# B&R Automation Studio project HealthCareDemo (part 2)

#### Router6D.fun - Exported functions and function blocks
```iecst
FUNCTION_BLOCK rl6dRouterMan (*Router manager*)
	VAR_INPUT
		Assembly : REFERENCE TO Mc6DAssemblyType; (*Assembly to manage shuttles on*)
		UserDataSize : UDINT; (*Size of the user data*)
		Enable : BOOL; (*Enable shuttle routing*)
	END_VAR
	VAR_OUTPUT
		Busy : BOOL; (*The function block is busy and must continue to be called*)
		Active : BOOL; (*The function block is active*)
		Error : BOOL; (*An error occurred*)
		ErrorID : DINT; (*Error that occurred*)
		Router : rl6dRouterType; (*Router handle*)
	END_VAR
	VAR
		Internal : rl6dRouterManInternalType; (*Internal data*)
	END_VAR
END_FUNCTION_BLOCK

FUNCTION_BLOCK rl6dRouterAddPathFromData (*Add a path from an array of positions*)
	VAR_INPUT
		Router : REFERENCE TO rl6dRouterType; (*Router to add path to*)
		DataAddress : UDINT; (*Pointer to array of rl6dPositionType*)
		DataSize : UDINT; (*Size of the array of positions in Bytes*)
		Name : STRING[255]; (*Name of the path*)
		Execute : BOOL; (*Add the path*)
	END_VAR
	VAR_OUTPUT
		Busy : BOOL; (*The function block is busy and must continue to be called*)
		Path : rl6dPathType; (*Path handle*)
		Done : BOOL; (*The path has been created*)
		Error : BOOL; (*An error occurred*)
		ErrorID : DINT; (*Error that occurred*)
	END_VAR
	VAR
		Internal : rl6dRouterAddPathInternalType; (*Internal data*)
	END_VAR
END_FUNCTION_BLOCK

FUNCTION_BLOCK rl6dPathGetData (*Get a path to an array of positions*)
	VAR_INPUT
		Path : REFERENCE TO rl6dPathType; (*Path handle*)
		DataAddress : UDINT; (*Pointer to array of rl6dPositionType*)
		DataSize : UDINT; (*Size of the array of positions in Bytes*)
		Execute : BOOL; (*Get the path*)
	END_VAR
	VAR_OUTPUT
		Busy : BOOL; (*The function block is busy and must continue to be called*)
		PathDataSize : UDINT; (*Actual size of path data*)
		Done : BOOL; (*The path has been created*)
		Error : BOOL; (*An error occurred*)
		ErrorID : DINT; (*Error that occurred*)
	END_VAR
	VAR
		Internal : rl6dGetPathInternalType; (*Internal data*)
	END_VAR
END_FUNCTION_BLOCK

FUNCTION_BLOCK rl6dRouterAddDestination (*Add a path from an array of positions*)
	VAR_INPUT
		Router : REFERENCE TO rl6dRouterType; (*Router to add destination to*)
		EntryPath : REFERENCE TO rl6dPathType; (*Optional reference to the destination entry path*)
		ExitPath : REFERENCE TO rl6dPathType; (*Optional reference to the destination exit path*)
		Position : rl6dPositionType; (*Position of the destination*)
		Name : STRING[255]; (*Name of the destination*)
		Execute : BOOL; (*Add the destination*)
	END_VAR
	VAR_OUTPUT
		Busy : BOOL; (*The function block is busy and must continue to be called*)
		Destination : rl6dDestinationType; (*Destination handle*)
		Done : BOOL; (*The destination has been created*)
		Error : BOOL; (*An error occurred*)
		ErrorID : DINT; (*Error that occurred*)
	END_VAR
	VAR
		Internal : rl6dRouterAddPathInternalType; (*Internal data*)
	END_VAR
END_FUNCTION_BLOCK

FUNCTION_BLOCK rl6dDestAddRecoveryPosFromData (*Add recovery positions from an array of positions*)
	VAR_INPUT
		Destination : REFERENCE TO rl6dDestinationType; (*Destination to add recovery points to*)
		DataAddress : UDINT; (*Pointer to array of rl6dPositionType*)
		DataSize : UDINT; (*Size of the array of positions in Bytes*)
		Execute : BOOL; (*Add the recovery points*)
	END_VAR
	VAR_OUTPUT
		Busy : BOOL; (*The function block is busy and must continue to be called*)
		Done : BOOL; (*The path has been created*)
		Error : BOOL; (*An error occurred*)
		ErrorID : DINT; (*Error that occurred*)
	END_VAR
	VAR
		Internal : rl6dDestAddRecPosInternalType; (*Internal data*)
	END_VAR
END_FUNCTION_BLOCK

FUNCTION_BLOCK rl6dDestinationSetWaypoint (*Set the waypoint of the destination*)
	VAR_INPUT
		Destination : REFERENCE TO rl6dDestinationType; (*Destination to set waypoint*)
		Waypoint : REFERENCE TO rl6dWaypointType; (*Waypoint to set*)
		Execute : BOOL; (*Set the next waypoint on a rising edge*)
	END_VAR
	VAR_OUTPUT
		Busy : BOOL; (*The function block is busy and must continue to be called*)
		Done : BOOL; (*The waypoint has been set*)
		Error : BOOL; (*An error occurred*)
		ErrorID : DINT; (*Error that occurred*)
	END_VAR
	VAR
		Internal : rl6dDestSetWaypntInternalType; (*Internal data*)
	END_VAR
END_FUNCTION_BLOCK

FUNCTION_BLOCK rl6dRouterAddWaypoint (*Add a waypoint from a position*)
	VAR_INPUT
		Router : REFERENCE TO rl6dRouterType; (*Router to add waypoint to*)
		Position : rl6dPositionType; (*Position of waypoint*)
		Name : STRING[255]; (*Name of waypoint*)
		Execute : BOOL; (*Add waypoint on rising edge*)
	END_VAR
	VAR_OUTPUT
		Busy : BOOL; (*The function block is busy and must continue to be called*)
		Waypoint : rl6dWaypointType; (*Waypoint handle*)
		Done : BOOL; (*The waypoint has been created*)
		Error : BOOL; (*An error occurred*)
		ErrorID : DINT; (*Error that occurred*)
	END_VAR
	VAR
		Internal : rl6dRouterAddWaypntInternalType; (*Internal data*)
	END_VAR
END_FUNCTION_BLOCK

FUNCTION_BLOCK rl6dWaypointAddDestination (*Add Destination to Waypoint*)
	VAR_INPUT
		Waypoint : REFERENCE TO rl6dWaypointType; (*Waypoint to add destination to*)
		Destination : REFERENCE TO rl6dDestinationType; (*Destination to add to waypoint*)
		DeparturePath : REFERENCE TO rl6dPathType; (*Optional departure path to follow when leaving waypoint for destination*)
		Execute : BOOL; (*Add the destination*)
	END_VAR
	VAR_OUTPUT
		Busy : BOOL; (*The function block is busy and must continue to be called*)
		Done : BOOL; (*The Destination has been added to the Waypoint*)
		Error : BOOL; (*An error occurred*)
		ErrorID : DINT; (*Error that occurred*)
	END_VAR
	VAR
		Internal : rl6dWaypointAddDestInternalType; (*Internal data*)
	END_VAR
END_FUNCTION_BLOCK

FUNCTION_BLOCK rl6dWaypointSetNextWaypoint (*Set the next waypoint of the target waypoint*)
	VAR_INPUT
		Waypoint : REFERENCE TO rl6dWaypointType; (*Waypoint to set next waypoint of*)
		NextWaypoint : REFERENCE TO rl6dWaypointType; (*Next waypoint*)
		Execute : BOOL; (*Set the next waypoint on a rising edge*)
	END_VAR
	VAR_OUTPUT
		Busy : BOOL; (*The function block is busy and must continue to be called*)
		Done : BOOL; (*The next waypoint has been set*)
		Error : BOOL; (*An error occurred*)
		ErrorID : DINT; (*Error that occurred*)
	END_VAR
	VAR
		Internal : rl6dWaypntSetWaypntInternalType; (*Internal data*)
	END_VAR
END_FUNCTION_BLOCK

FUNCTION_BLOCK rl6dRouterAddShFromAsm (*Add shuttles from the assembly*)
	VAR_INPUT
		Router : REFERENCE TO rl6dRouterType; (*Router to add shuttles from assembly to*)
		Execute : BOOL; (*Add shuttles*)
	END_VAR
	VAR_OUTPUT
		Busy : BOOL; (*The function block is busy and must continue to be called*)
		Done : BOOL; (*The shuttles have been added*)
		NumShuttles : UDINT; (*Number of shuttles found on the assembly*)
		Error : BOOL; (*An error occurred*)
		ErrorID : DINT; (*Error that occurred*)
	END_VAR
	VAR
		Internal : rl6dRtrAddShFromAsmInternalType; (*Internal data*)
	END_VAR
END_FUNCTION_BLOCK

FUNCTION_BLOCK rl6dRouterExecuteRecovery (*Execute recovery of shuttles*)
	VAR_INPUT
		Router : REFERENCE TO rl6dRouterType; (*Router to add shuttles from assembly to*)
		Velocity : REAL; (*Recovery Velocity*)
		Acceleration : REAL; (*Recovery Acceleration*)
		Mode : rl6dRecoverModeEnum; (*Mode to use when recovering*)
		Execute : BOOL; (*Add shuttles*)
	END_VAR
	VAR_OUTPUT
		Busy : BOOL; (*The function block is busy and must continue to be called*)
		Done : BOOL; (*The shuttles have been added*)
		Error : BOOL; (*An error occurred*)
		ErrorID : DINT; (*Error that occurred*)
	END_VAR
	VAR
		Internal : rl6dRtrAddShFromAsmInternalType; (*Internal data*)
	END_VAR
END_FUNCTION_BLOCK

FUNCTION_BLOCK rl6dDestinationMonitor (*Monitor destination for shuttles*)
	VAR_INPUT
		Destination : REFERENCE TO rl6dDestinationType; (*Destination to monitor*)
		Enable : BOOL; (*Enable monitoring*)
		AcknowledgeShuttle : BOOL; (*Acknowledge current shuttle*)
	END_VAR
	VAR_OUTPUT
		Busy : BOOL; (*The function block is busy and must continue to be called*)
		Valid : BOOL; (*Outputs are valid*)
		ShuttlePresent : BOOL; (*A shuttle is present at the destination*)
		ShuttleID : UINT; (*Shuttle ID*)
		RouterShuttle : rl6dShuttleType; (*Shuttle for use with router system*)
		Mc6DShuttle : Mc6DShuttleType; (*Shuttle for use with mapp 6D*)
		Error : BOOL; (*An error occurred*)
		ErrorID : DINT; (*Error that occurred*)
	END_VAR
	VAR
		Internal : rl6dDestinationMonInternalType; (*Internal data*)
	END_VAR
END_FUNCTION_BLOCK

FUNCTION_BLOCK rl6dShuttleMoveDestination (*Move shuttle to destination*)
	VAR_INPUT
		RouterShuttle : REFERENCE TO rl6dShuttleType; (*Shuttle to control*)
		Destination : REFERENCE TO rl6dDestinationType; (*Destination to move to*)
		Waypoint : REFERENCE TO rl6dWaypointType; (*Optional waypoint to override the waypoint specified by the previous destination*)
		Velocity : REAL; (*Velocity of shuttle movement*)
		Acceleration : REAL; (*Acceleration of shuttle movement*)
		Execute : BOOL; (*Start moving shuttle to destination*)
	END_VAR
	VAR_OUTPUT
		Busy : BOOL; (*The function block is busy and must continue to be called*)
		Active : BOOL; (*Move is active*)
		Aborted : BOOL; (*Move has been aborted*)
		Done : BOOL; (*Move has completed*)
		Error : BOOL; (*An error occurred*)
		ErrorID : DINT; (*Error that occurred*)
	END_VAR
	VAR
		Internal : rl6dShMoveDestInternalType; (*Internal data*)
	END_VAR
END_FUNCTION_BLOCK

FUNCTION_BLOCK rl6dShCopyUserData (*Copy shuttle user data asynchronously*)
	VAR_INPUT
		RouterShuttle : REFERENCE TO rl6dShuttleType; (*Shuttle to copy user data*)
		Mode : rl6dShCopyUserDataModeEnum; (*Mode of copy user data*)
		DataAddress : UDINT; (*Address of data to copy*)
		DataSize : UDINT; (*Start moving shuttle to destination*)
		Execute : BOOL; (*Copy user data*)
	END_VAR
	VAR_OUTPUT
		Busy : BOOL; (*The function block is busy and must continue to be called*)
		Done : BOOL; (*Move has completed*)
		SizeCopied : UDINT; (*Size of the data copied*)
		Error : BOOL; (*An error occurred*)
		ErrorID : DINT; (*Error that occurred*)
	END_VAR
	VAR
		Internal : rl6dShCopyUserDataInternalType; (*Internal Data*)
	END_VAR
END_FUNCTION_BLOCK

FUNCTION rl6dShCopyUserDataSync : DINT (*Copy shuttle user data synchronously*)
	VAR_INPUT
		RouterShuttle : rl6dShuttleType; (*Shuttle to copy user data*)
		Mode : rl6dShCopyUserDataModeEnum; (*Mode of copy*)
		DataAddress : UDINT; (*Data address*)
		DataSize : UDINT; (*Data size*)
	END_VAR
END_FUNCTION
```

#### CheckRef.hpp - Check Reference Headers
```cpp
#ifndef __RL6D_CHECK_REF_H__
#define __RL6D_CHECK_REF_H__

#include <Router.hpp>
#include <SemMan.hpp>
#include <Destination.hpp>
#include <DestinationIf.hpp>
#include <Path.hpp>
#include <Shuttle.hpp>
#include <ShuttleIf.hpp>

//Forward Declarations
class Router;
class SemMan;
class RouterSem;
class Destination;
class DestinationIf;
class Path;
class Shuttle;
class ShuttleIf;

DINT check_null_pointer(UDINT reference);

DINT check_router_reference(rl6dRouterType* reference);

DINT check_sem_man_reference(UDINT reference);

DINT check_router_sem_reference(UDINT reference);

DINT check_destination_reference(rl6dDestinationType* reference);

DINT check_destination_if_reference(UDINT reference);

DINT check_path_reference(rl6dPathType* reference);

DINT check_waypoint_reference(rl6dWaypointType* reference);

DINT check_shuttle_reference(rl6dShuttleType* reference);

DINT check_shuttle_if_reference(UDINT reference);

#endif
```

#### Logging.hpp - Logging Headers
```cpp
#ifndef __RL6D_LOGGING_H__
#define __RL6D_LOGGING_H__

#include <Router6D.h>
#include <string>
#include <cstring>

extern plcstring router_6d_log_name [];

bool log_routed_move_start(UINT shuttle, std::string destination);

bool log_direct_move_start(UINT shuttle, std::string destination);

bool log_destination_arrival(UINT shuttle, std::string destination);

bool log_destination_update(UINT shuttle, std::string destination);

bool log_path_start(UINT shuttle, std::string path);

bool log_waypoint_move(UINT shuttle, std::string waypoint);

bool log_routed_move_waypoint(UINT shuttle, std::string destination, std::string waypoint);

bool log_asm_get_sh_start(void);

bool log_asm_get_sh_done(UINT shuttles);

bool log_asm_recovery_start(rl6dRecoverModeEnum mode);

bool log_asm_recovery_done(void);

bool log_asm_sh_assignment(UINT shuttle, std::string destination);

bool log_sh_error(UINT shuttle, DINT error);

bool log_asm_get_sh_error(DINT error);

bool log_move_in_plane_error(DINT error);

#endif
```

#### Router.hpp - Router Headers
```cpp
#ifndef __RL6D_ROUTER_H__
#define __RL6D_ROUTER_H__

#include <memory>
#include <algorithm>
#include <cstring>

#include <CheckRef.hpp>
#include <Path.hpp>
#include <Waypoint.hpp>
#include <Shuttle.hpp>
#include <SemMan.hpp>
#include <Logging.hpp>

struct RouterCmd{
    bool add_sh_from_asm = 0;
    bool recover_shuttles = 0;
    rl6dRecoverModeEnum recover_shuttles_mode = rl6dRECOVER_MODE_BASIC;
    bool error_reset = 0;
};

struct RouterStatus{
    bool cmd_ready = 0;
    bool done = 0;
    bool error = 0;
    DINT error_id = 0;
};

struct ShDestAssignment{
    std::shared_ptr<Shuttle> shuttle;
    std::shared_ptr<Destination> destination;
};

/**
 \brief A Router manages shuttles to destinations
*/
class Router : public SemManBase{
    public:
    //! constructor for the Router
    Router(Mc6DAssemblyType* assembly, UDINT user_data_size);

    //! destructor for the Router
    ~Router(void);

    // members

    // methods
    //! Get the Router Type ID
    UDINT get_type_id(void);
    //! Create a new path
    std::shared_ptr<Path> create_path(std::string name, std::shared_ptr<RouterSem> router_sem);
    //! Delete a path
    void delete_path(std::shared_ptr<Path>);
    //! Get a path by name
    std::shared_ptr<Path> get_path_by_name(std::string name);
    //! Create a destination
    std::shared_ptr<Destination> create_destination(std::string name, std::shared_ptr<RouterSem> router_sem, rl6dPositionType position, std::shared_ptr<Path> path_in, std::shared_ptr<Path> path_out);
    //! Create a waypoint
    std::shared_ptr<Waypoint> create_waypoint(std::string name, std::shared_ptr<RouterSem> router_sem, rl6dPositionType position);
    //! Add a shuttle
    std::shared_ptr<Shuttle> add_shuttle(Mc6DShuttleType shuttle, std::shared_ptr<RouterSem> router_semaphore, UINT shuttle_id);
    //! Remove a shuttle
    void delete_shuttle(Mc6DShuttleType shuttle);
    //! Acquire path semaphore
    bool acquire_path_semaphore(void);
    //! Release path semaphore
    void release_path_semaphore(void);
    //! Acquire waypoint semaphore
    bool acquire_waypoint_semaphore(void);
    //! Release waypoint semaphore
    void release_waypoint_semaphore(void);
    //! Acquire shuttle semaphore
    bool acquire_shuttle_semaphore(void);
    //! Release shuttle semaphore
    void release_shuttle_semaphore(void);
    //! Acquire destination semaphore
    bool acquire_destination_semaphore(void);
    //! Release destination semaphore
    void release_destination_semaphore(void);
    //! Acquire command semaphore
    bool acquire_cmd_semaphore(void);
    //! Release command semaphore
    void release_cmd_semaphore(void);
    //! Set add shuttles from assembly
    void set_add_sh_from_asm();
    //! Reset add shuttles from assembly
    void reset_add_sh_from_asm(void);
    //! Set recover shuttles
    void set_recover_shuttles(rl6dRecoverModeEnum mode, REAL velocity, REAL acceleration);
    //! Reset recover shuttles
    void reset_recover_shuttles(void);
    //! Reset router errors
    void set_error_reset(void);
    //! get the number of shuttles found on the assembly
    UINT get_num_asm_sh(void);
    //! Get ready status
    bool get_cmd_ready(void);
    //! Get Done status
    bool get_done(void);
    //! Get error status
    bool get_error(void);
    //! Get error ID
    DINT get_error_id(void);
    //! Get initialized status
    bool get_initialized(void);
    //! Cyclic execution
    void cyclic(void);

    private:

    enum _state_enum
    {
        STATE_INIT,
        STATE_EVENT_LOG_CREATE,
        STATE_WAIT_SEM,
        STATE_CREATE_PATH_SEM,
        STATE_CREATE_WAYPOINT_SEM_READY,
        STATE_CREATE_WAYPOINT_SEM,
        STATE_CREATE_SHUTTLE_SEM_READY,
        STATE_CREATE_SHUTTLE_SEM,
        STATE_CREATE_DESTINATION_SEM_READY,
        STATE_CREATE_DESTINATION_SEM,
        STATE_CREATE_CMD_SEM_READY,
        STATE_CREATE_CMD_SEM,
        STATE_ACTIVE,
        STATE_ADD_SH_ASM,
        STATE_ADD_SH_ASM_SEM,
        STATE_ADD_SH_ASM_NEXT,
        STATE_ADD_SH_ASM_DONE,
        STATE_RECOVER_SHUTTLES_GET_DEST,
        STATE_RECOVER_SHUTTLES_GET_POS,
        STATE_RECOVER_SHUTTLES_ASSIGN,
        STATE_RECOVER_SHUTTLES,
        STATE_RECOVER_DESTINATION,
        STATE_RECOVER_DESTINATION_WAIT,
        STATE_RECOVER_SHUTTLES_DONE,
        STATE_ERROR
    };

    //! type identifier to ensure that pointer is valid
    UDINT _type_id = rl6dROUTER_TYPE_ID;
    //! state
    _state_enum _state = STATE_INIT;
    //! the list of paths that are part of the router
    std::vector<std::shared_ptr<Path>> _paths;
    //! the list of waypoints that are part of the router
    std::vector<std::shared_ptr<Waypoint>> _waypoints;
    //! the list of destinations that are part of the router
    std::vector<std::shared_ptr<Destination>> _destinations;
    //! the list of destinations to recover to
    std::vector<std::shared_ptr<Destination>> _recovery_destinations;
    //! current detination recovered shuttles are being assigned
    std::shared_ptr<Destination> _current_recovery_destination;
    //! current positions recovered shuttles are being assigned
    std::vector<rl6dPositionType> _current_recovery_positions;
    //! the list of shuttles that are part of the router
    std::vector<std::shared_ptr<Shuttle>> _shuttles;
    //! the list of shuttles to recover
    std::vector<std::shared_ptr<Shuttle>> _recovery_shuttles;
    //! current shuttle being recovered
    std::shared_ptr<Shuttle> _current_recovery_shuttle;
    //! current recovery index
    unsigned int _current_recovery_index = 0;
    //! current recovery position
    rl6dPositionType _current_recovery_position;
    //! the list of final recovery moves to make
    std::vector<ShDestAssignment> _shuttle_destination_assignment;
    //! current recovery shuttle interface
    std::shared_ptr<ShuttleIf> _current_recovery_shuttle_interface;
    //! the list of recovery shuttle interfaces
    std::vector<std::shared_ptr<ShuttleIf>> _shuttle_recovery_interfaces;
    //! Path semaphore
    std::shared_ptr<RouterSem> _path_semaphore;
    //! Waypoint semaphore
    std::shared_ptr<RouterSem> _waypoint_semaphore;
    //! Destination semaphore
    std::shared_ptr<RouterSem> _destination_semaphore;
    //! Shuttle semaphore
    std::shared_ptr<RouterSem> _shuttle_semaphore;
    //! Command semaphore
    std::shared_ptr<RouterSem> _command_semaphore;
    //! Router commands
    RouterCmd _cmd;
    //! Router status
    RouterStatus _status;
    //! Get shuttles from assembly
    struct MC_BR_AsmGetShuttle_Acp6D _asm_get_shuttle;
    //! Recover shuttles on assembly
    struct MC_BR_MoveInPlaneAsync_Acp6D _move_in_plane_async;
    //! Recorded number of shuttles remaining from assembly
    UDINT _old_remaining_count = 0;
    //! Recorded number of shuttles found on the assembly
    UDINT _asm_shuttles = 0;
    //! Newly created semaphore
    std::shared_ptr<RouterSem> _created_semaphore;
    //! Flag that initial semaphore creation is complete
    bool _router_sem_complete = 0;
    //! User data size for all shuttles
    UDINT _user_data_size;
    //! Initialization is complete
    bool _init_done = 0;
    //! Error
    bool _error = 0;
    //! Error ID
    DINT _error_id = ERR_OK;
    //EventLog Create
    struct ArEventLogCreate _ar_event_log_create;

};

#endif
```

#### SemMan.hpp - SemMan Headers
```cpp
#ifndef __RL6D_SEMMAN_H__
#define __RL6D_SEMMAN_H__

#include <memory>
#include <vector>
#include <algorithm>
#include <cstring>

#include <Router6D.h>

/**
 \brief A RouterSem contains a semaphore
*/
class RouterSem : public std::enable_shared_from_this<RouterSem>{
    public:
    //! constructor for the RouterSem
    RouterSem(UDINT semaphore);

    //! destructor for the RouterSem
    ~RouterSem(void);

    // members

    // methods
    //! Get the RouterSem Type ID
    UDINT get_type_id(void);
    //! Get the semaphore ident
    UDINT get_semaphore_ident(void);
    //! Delete this semaphore
    void set_delete(void);
    //! Check if this semaphore is to be deleted
    bool get_delete(void);
    //! Acquire the semaphore
    bool sem_acquire(void);
    //! Release the semaphore
    void sem_release(void);
    //! Get existing shared pointer
    std::shared_ptr<RouterSem> get_shared_ptr(void);

    private:

    //! type identifier to ensure that pointer is valid
    UDINT _type_id = rl6dROUTER_SEM_TYPE_ID;
    //! Semaphore to access
    UDINT _sem;
    //! Flag if this semaphore is to be deleted
    bool _delete = 0;

};

/**
 \brief A RouterSemBase gives a derived class the public methods and attributes to interface with the contained RouterSem
*/
class RouterSemBase{
    public:
    //! constructor for the RouterSem
    RouterSemBase(std::shared_ptr<RouterSem>);

    //! destructor for the RouterSem
    ~RouterSemBase(void);

    // members

    // methods
    //! Acquire the semaphore
    bool sem_acquire(void);
    //! Release the semaphore
    void sem_release(void);

    protected:

    //! Router semaphore
    std::shared_ptr<RouterSem> _router_semaphore;

};

struct SemManCmd{
    bool create_sem = 0;
    bool delete_all = 0;
};

struct SemManStatus{
    bool cmd_ready = 0;
    bool done = 0;
    bool error = 0;
    DINT error_id = 0;
};

/**
 \brief A SemMan mangages semaphores
*/
class SemMan{
    public:
    //! constructor for the SemMan
    SemMan(void);

    //! destructor for the SemMan
    ~SemMan(void);

    // members

    // methods
    //! Get the SemMan Type ID
    UDINT get_type_id(void);
    //! Create a new semaphore
    void set_create_sem(void);
    //! Reset creating a new semaphore
    void reset_create_sem(void);
    //! Return the newly created semaphore
    std::shared_ptr<RouterSem> get_created_sem(void);
    //! Get Done status
    bool get_done(void);
    //! Get Command Ready status
    bool get_cmd_ready(void);
    //! Get Error status
    bool get_error(void);
    //! Get Error ID
    DINT get_error_id(void);
    //! Delete a semaphore
    void delete_sem(UDINT);
    //! Acquire the semaphore to use other methods
    bool sem_acquire(void);
    //! Release the semaphore
    void sem_release(void);
    //! Get if the initialization is done
    bool get_initialized(void);
    //! Cyclic execution
    void cyclic(void);

    private:

    enum _state_enum
    {
        STATE_START,
        STATE_INIT,
        STATE_IDLE,
        STATE_CREATE_SEM,
        STATE_CREATE_SEM_DONE,
        STATE_DELETE_SEM,
        STATE_DELETE_ALL_SEM,
        STATE_DELETE_ALL_SEM_NEXT,
        STATE_DELETE_ALL_SEM_LAST,
        STATE_DELETE_ALL_SEM_DONE
    };

    //! type identifier to ensure that pointer is valid
    UDINT _type_id = rl6dSEM_MAN_TYPE_ID;
    //! state
    _state_enum _state = STATE_START;
    //! Semaphore to access manager
    UDINT _sem;
    //! Initialization is complete
    bool _init_done = 0;
    //! Commands
    SemManCmd _cmd;
    //! Status
    SemManStatus _status;
    //! Created semaphore
    std::shared_ptr<RouterSem> _created_semaphore;
    //! the list of semaphores being managed
    std::vector<std::shared_ptr<RouterSem>> _semaphores;
    //! Redo so that the iterator is not needed
    std::vector<std::shared_ptr<RouterSem>>::iterator _sem_iterator;
    //! semaphore generator
    struct SemCreate _create_semaphore;
    //! semaphore destructor
    struct SemDelete _delete_semaphore;

};

/**
 \brief A SemManBase gives a derived class the public methods and attributes to interface with the contained SemMan
*/
class SemManBase{
    public:
    //! constructor for the SemManBase
    SemManBase(void);

    //! destructor for the SemManBase
    ~SemManBase(void);

    // members

    // methods
    //! Create a new semaphore
    void set_create_sem(void);
    //! Reset creating a new semaphore
    void reset_create_sem(void);
    //! Return the newly created semaphore
    std::shared_ptr<RouterSem> get_created_sem(void);
    //! Get Done status
    bool get_sem_done(void);
    //! Get Command Ready status
    bool get_sem_cmd_ready(void);
    //! Get Error status
    bool get_sem_error(void);
    //! Get Error ID
    DINT get_sem_error_id(void);
    //! Acquire the semaphore to use other methods
    bool sem_acquire(void);
    //! Release the semaphore
    void sem_release(void);

    protected:

    //! SemMan
    SemMan _semaphore_manager;

};

#endif
```

#### Destination.hpp - Destination Headers
```cpp
#ifndef __RL6D_DESTINATION_H__
#define __RL6D_DESTINATION_H__

#include <memory>
#include <algorithm>
#include <string>
#include <vector>
#include <Router6D.h>

#include <Shuttle.hpp>
#include <Path.hpp>
#include <DestinationIf.hpp>
#include <Waypoint.hpp>

//Forward Declarations
class DestinationIf;
class Shuttle;
class Waypoint;

/**
 \brief A Destination is a position that a shuttle can travel to and can notify of its arrival
*/
class Destination: public RouterSemBase, public std::enable_shared_from_this<Destination>{
    public:
    //! constructor for the Destination
    Destination(std::string name, std::shared_ptr<RouterSem> router_sem);
    Destination(std::string name, std::shared_ptr<RouterSem> router_sem, rl6dPositionType position);
    Destination(std::string name, std::shared_ptr<RouterSem> router_sem, rl6dPositionType position, std::shared_ptr<Path> path_in, std::shared_ptr<Path> path_out);

    //! destructor for the Destination
    ~Destination(void);

    // members

    // methods
    //! Get the destination type ID
    UDINT get_type_id(void);
    //! Get the destination name
    std::string get_name(void);
    //! Get the destination position
    rl6dPositionType get_position(void);
    //! Get the recovery positions
    std::vector<rl6dPositionType> get_recovery_positions(void);
    //! Set the destination position
    void set_position(rl6dPositionType position);
    //! Get the destination path in
    std::shared_ptr<Path> get_path_in(void);
    //! Set the destination path in
    void set_path_in(std::shared_ptr<Path> path);
    //! Clear the destination path in
    void clear_path_in(void);
    //! Get the destination path out
    std::shared_ptr<Path> get_path_out(void);
    //! Set the destination path out
    void set_path_out(std::shared_ptr<Path> path);
    //! Clear the destination path out
    void clear_path_out(void);
    //! Add recovery position
    void add_recovery_position(rl6dPositionType position);
    //! Create interface
    std::shared_ptr<DestinationIf> create_interface(void);
    //! Set waypoint
    void set_waypoint(std::weak_ptr<Waypoint> waypoint);
    //! Get waypoint
    std::weak_ptr<Waypoint> get_waypoint(void);
    //! Reset waypoint
    void reset_waypoint(void);
    //! Set shuttle present
    void set_shuttle_present(std::weak_ptr<Shuttle> shuttle);
    //! Get existing shared pointer
    std::shared_ptr<Destination> get_shared_ptr(void);
    //! Cyclic runtime
    void cyclic(void);

    private:

    //! destination position
    rl6dPositionType _position;
    //! type identifier to ensure that pointer is valid
    UDINT _type_id = rl6dDESTINATION_TYPE_ID;
    //! name of the destination
    std::string _name;
    //! path in
    std::shared_ptr<Path> _path_in;
    //! path out
    std::shared_ptr<Path> _path_out;
    //! default waypoint
    std::weak_ptr<Waypoint> _waypoint;
    //! recovery points
    std::vector<rl6dPositionType> _recovery_positions;
    //! the list of destination interfaces that are part of the destination
    std::vector<std::shared_ptr<DestinationIf>> _interfaces;
    //! shuttle present at destination
    std::weak_ptr<Shuttle> _shuttle;
    //! shuttle present status
    bool _shuttle_present = 0;

};

#endif
```

#### DestinationIf.hpp - DestinationIf Headers
```cpp
#ifndef __RL6D_DESTINATION_IF_H__
#define __RL6D_DESTINATION_IF_H__

#include <memory>

#include <Router6D.h>
#include <Shuttle.hpp>

class Shuttle; //Forward Declaration

/**
 \brief A DestinationIf is an interface that can be monitored for shuttles
*/
class DestinationIf: public std::enable_shared_from_this<DestinationIf>{
    public:
    //! constructor for the DestinationIf
    DestinationIf(void);

    //! destructor for the DestinationIf
    ~DestinationIf(void);

    // members

    // methods
    //! Get the DestinationIf type ID
    UDINT get_type_id(void);
    //! Get existing shared pointer
    std::shared_ptr<DestinationIf> get_shared_ptr(void);
    //! Set shuttle status
    void set_shuttle_present(std::weak_ptr<Shuttle> shuttle);
    //! Get shuttle status
    bool shuttle_is_present(void);
    //! Get currently present shuttle
    std::weak_ptr<Shuttle> get_shuttle_present(void);
    //! Acknowledge shuttle present
    void acknowledge_shuttle(void);
    //! Set interface for deletion
    void set_delete(void);
    //! Check interface for deletion
    bool get_delete(void);

    private:

    //! type identifier to ensure that pointer is valid
    UDINT _type_id = rl6dDESTINATION_IF_TYPE_ID;
    //! Destination status of shuttle present
    bool _shuttle_present = 0;
    //! Shuttle present at Destination
    std::weak_ptr<Shuttle> _shuttle;
    //! Interface can be deleted
    bool _delete = 0;

};

#endif
```

#### Path.hpp - Path Headers
```cpp
#ifndef __RL6D_PATH_H__
#define __RL6D_PATH_H__

#include <string>
#include <vector>
#include <Router6D.h>
#include <SemMan.hpp>

/**
 \brief A Path is a vector of positions that the shuttle can travel along bust cannot leave
*/
class Path : public RouterSemBase, public std::enable_shared_from_this<Path>{
    public:
    //! constructor for the Path
    Path(std::string name, std::shared_ptr<RouterSem> router_sem);

    //! destructor for the Path
    ~Path(void);

    // members

    // methods
    //! Get the path type ID
    UDINT get_type_id(void);
    //! Get the path name
    std::string get_name(void);
    //! Add a position to the vector
    void add_position(rl6dPositionType position);
    //! Get position vector
    std::vector<rl6dPositionType> get_positions(void);
    //! Get existing shared pointer
    std::shared_ptr<Path> get_shared_ptr(void);

    private:

    //! the list of positions that are part of the path
    std::vector<rl6dPositionType> _positions;
    //! type identifier to ensure that pointer is valid
    UDINT _type_id = rl6dPATH_TYPE_ID;
    //! name of the path
    std::string _name;

};

#endif
```

#### Waypoint.hpp - Waypoint Headers
```cpp
#ifndef __RL6D_WAYPOINT_H__
#define __RL6D_WAYPOINT_H__

#include <Router6D.h>
#include <Path.hpp>
#include <Destination.hpp>

class Destination; //Forward declaration

struct WaypointDestination{
    std::shared_ptr<Destination> destination;
    std::shared_ptr<Path> departure_path;
};

/**
 \brief A Waypoint is a position that the shuttle will go through on its way to a destination, if defined
*/
class Waypoint : public RouterSemBase, public std::enable_shared_from_this<Waypoint>{
    public:
    //! constructor for the Waypoint
    Waypoint(std::string name, std::shared_ptr<RouterSem> router_sem);
    Waypoint(std::string name, std::shared_ptr<RouterSem> router_sem, rl6dPositionType position);

    //! destructor for the Waypoint
    ~Waypoint(void);

    // members

    // methods
    //! Get the waypoint type ID
    UDINT get_type_id(void);
    //! Get the waypoint name
    std::string get_name(void);

    //! Add an accessible destination to the waypoint
    void add_destination(std::shared_ptr<Destination> destination, std::shared_ptr<Path> departure_path);
    //! Check if a destination is accessible
    bool check_destination_accessible(std::shared_ptr<Destination> destination);
    //! Get destination departure path
    std::shared_ptr<Path> get_destination_departure_path(std::shared_ptr<Destination> destination);
    //! Get destination vector
    std::vector<WaypointDestination> get_destinations(void);
    //! Get position
    rl6dPositionType get_position(void);
    //! Get existing shared pointer
    std::shared_ptr<Waypoint> get_shared_ptr(void);
    //! Get next waypoint
    std::weak_ptr<Waypoint> get_next_waypoint(void);
    //! Set next waypoint
    void set_next_waypoint(std::weak_ptr<Waypoint> waypoint);
    //! Reset next waypoint
    void reset_next_waypoint(void);

    private:

    //! the next waypoint
    std::weak_ptr<Waypoint> _next_waypoint;
    //! the list of destinations accessible from the waypoint
    std::vector<WaypointDestination> _destinations;
    //! type identifier to ensure that pointer is valid
    UDINT _type_id = rl6dWAYPOINT_TYPE_ID;
    //! name of the waypoint
    std::string _name;
    //! position of the waypoint
    rl6dPositionType _position;

};

#endif
```

#### Shuttle.hpp - Shuttle Headers
```cpp
#ifndef __RL6D_SHUTTLE_H__
#define __RL6D_SHUTTLE_H__

#include <Router6D.h>
#include <McAcp6D.h>
#include <memory>
#include <vector>
#include <algorithm>
#include <cstring>

#include <Destination.hpp>
#include <Waypoint.hpp>
#include <Path.hpp>
#include <ShuttleIf.hpp>
#include <Logging.hpp>

class Destination; //Forward Declaration
class Waypoint; //Forward Declaration
class ShuttleIf; //Forward Declaration

struct ReadUserDataResult{
    char* value;
    UDINT size;
};

enum set_path_status_enum
{
    set_path_status_valid,
    set_path_status_invalid,
    set_path_status_wait_sem
};

enum routed_move_phase_enum
{
    ROUTED_MOVE_PHASE_EXIT_DEST_START,
    ROUTED_MOVE_PHASE_EXIT_DEST,
    ROUTED_MOVE_PHASE_WAYPOINT_START,
    ROUTED_MOVE_PHASE_WAYPOINT,
    ROUTED_MOVE_PHASE_DEPART_WAYPOINT_START,
    ROUTED_MOVE_PHASE_DEPART_WAYPOINT,
    ROUTED_MOVE_PHASE_ENTER_DEST_START,
    ROUTED_MOVE_PHASE_ENTER_DEST,
    ROUTED_MOVE_PHASE_DEST,
    ROUTED_MOVE_PHASE_ARRIVE
};

enum routed_move_event_enum
{
    ROUTED_MOVE_EVENT_NONE,
    ROUTED_MOVE_EVENT_PATH_START,
    ROUTED_MOVE_EVENT_WAYPOINT
};

struct RoutedMoveEvent{
    routed_move_event_enum event = ROUTED_MOVE_EVENT_NONE;
    std::shared_ptr<Path> path;
    std::weak_ptr<Waypoint> waypoint;
};

/**
 \brief A ShuttleRoutePositionGenerator outputs the positions on the shuttle route
*/
class ShuttleRoutePositionGenerator{
    public:
    //Constructor
    ShuttleRoutePositionGenerator(void);
    ShuttleRoutePositionGenerator(std::shared_ptr<Destination> previous_destination, std::shared_ptr<Destination> next_destination);
    ShuttleRoutePositionGenerator(std::shared_ptr<Destination> previous_destination, std::shared_ptr<Destination> next_destination, std::weak_ptr<Waypoint> route_waypoint);
    //Destructor
    ~ShuttleRoutePositionGenerator(void);

    //members

    //attributes
    rl6dPositionType position;
    RoutedMoveEvent event;

    //methods
    //! Increment the position along the route, return true if the route position has been incremented
    bool operator++(int);
    //! Update the destination
    void update_destination(std::shared_ptr<Destination> destination);
    void update_destination(std::shared_ptr<Destination> destination, std::weak_ptr<Waypoint> waypoint);
    //! Reset the position generator
    void reset(void);
    //! Get the current phase of the routed move
    routed_move_phase_enum get_phase(void);
    //! Get if the routed move is done
    bool get_done(void);

    private:

    //! Routing complete
    bool _done = 0;
    //! Set path, return set path status
    set_path_status_enum _set_path(std::shared_ptr<Path> path);
    //! Status of the exit path
    set_path_status_enum _exit_path_status = set_path_status_invalid;
    //! Status of the departure path
    set_path_status_enum _departure_path_status = set_path_status_invalid;
    //! Status of the entry path
    set_path_status_enum _entry_path_status = set_path_status_invalid;
    //! current waypoint
    std::weak_ptr<Waypoint> _current_waypoint;
    //! The phase of the routed motion
    routed_move_phase_enum _phase = ROUTED_MOVE_PHASE_EXIT_DEST_START;
    //! The previous destination the shuttle is going from
    std::shared_ptr<Destination>  _previous_destination;
    //! The next destination the shuttle is going to
    std::shared_ptr<Destination> _next_destination;
    //! The updated destination the shuttle needs to move to
    std::shared_ptr<Destination> _updated_destination;
    //! Route waypoint to use
    std::weak_ptr<Waypoint> _route_waypoint;
    //! path
    std::shared_ptr<Path> _path;
    //! path positions
    std::vector<rl6dPositionType> _path_positions;
    //! path iterator
    std::vector<rl6dPositionType>::iterator _path_iterator;
    //! Departure path
    std::shared_ptr<Path> _departure_path;

};

/**
 \brief A Shuttle controls an ACOPOS 6D shuttle
*/
class Shuttle : public RouterSemBase, public std::enable_shared_from_this<Shuttle>{
    public:
    //! constructor for the Shuttle
    Shuttle(Mc6DShuttleType shuttle, std::shared_ptr<RouterSem> router_sem, UDINT user_data_size, UINT _shuttle_id);

    //! destructor for the Shuttle
    ~Shuttle(void);

    // members

    // methods
    //! Get the shuttle type ID
    UDINT get_type_id(void);
    //! Get the shuttle ID
    UINT get_shuttle_id(void);
    //! Get the shuttle reference
    Mc6DShuttleType* get_shuttle_reference(void);
    //! Get the current destination
    std::shared_ptr<Destination> get_current_destination(void);
    //! Get the previous destination
    std::shared_ptr<Destination> get_previous_destination(void);
    //! Clear previous destination
    void clear_previous_destination(void);
    //! Create interface
    std::shared_ptr<ShuttleIf> create_interface(void);
    //! Get existing shared pointer
    std::shared_ptr<Shuttle> get_shared_ptr(void);
    //! Read User Data
    ReadUserDataResult read_user_data(void);
    //! Write User Data
    UDINT write_user_data(char* value, UDINT size);
    //! Cyclic runtime
    void cyclic(void);

    private:

    enum _state_enum
    {
        STATE_IDLE,
        STATE_ROUTED_MOVE_START,
        STATE_ROUTED_MOVE,
        STATE_ROUTED_MOVE_NEXT,
        STATE_DIRECT_MOVE,
    };

    //! Update shuttle interfaces
    bool _update_interfaces(void);
    //! Log events generated by the position generator
    void _log_event(RoutedMoveEvent event);
    //! type identifier to ensure that pointer is valid
    UDINT _type_id = rl6dSHUTTLE_TYPE_ID;
    //! 6D Shuttle ID
    UINT _shuttle_id;
    //! current interface
    std::shared_ptr<ShuttleIf> _current_interface;
    //! the list of shuttle interfaces that are part of the shuttle
    std::vector<std::shared_ptr<ShuttleIf>> _interfaces;
    //! The previous destination the shuttle is going from
    std::shared_ptr<Destination>  _previous_destination;
    //! The next destination the shuttle is going to
    std::shared_ptr<Destination> _next_destination;
    //! current state of cyclic execution
    _state_enum _state = STATE_IDLE;
    //! shuttle being managed
    Mc6DShuttleType _shuttle;
    //! move shuttle in plane
    struct MC_BR_MoveInPlane_Acp6D _move_in_plane;
    //! User Data
    std::unique_ptr<char[]> _user_data;
    //! User Data Size
    UDINT _user_data_size;
    //! Route position generator
    ShuttleRoutePositionGenerator _route_position_generator;
    //! Optional route waypoint
    std::weak_ptr<Waypoint> _optional_waypoint;

};

#endif
```

#### ShuttleIf.hpp - ShuttleIf Headers
```cpp
#ifndef __RL6D_SHUTTLE_IF_H__
#define __RL6D_SHUTTLE_IF_H__

#include <Router6D.h>

#include <Destination.hpp>
#include <Waypoint.hpp>

class Destination; //Forward Declaration
class Waypoint; //Forward Declaration

/**
 \brief A ShuttleIf is an interface that can be used to command shuttles
*/
class ShuttleIf : public std::enable_shared_from_this<ShuttleIf>{
    public:
    //! constructor for the ShuttleIf
    ShuttleIf(void);

    //! destructor for the ShuttleIf
    ~ShuttleIf(void);

    // members

    // methods
    //! Get the ShuttleIf type ID
    UDINT get_type_id(void);
    //! Issue move destination command
    void set_destination(std::shared_ptr<Destination> destination, REAL velocity, REAL acceleration);
    //! Issue move destination via waypoint command
    void set_destination_waypoint(std::shared_ptr<Destination> destination, std::weak_ptr<Waypoint> waypoint, REAL velocity, REAL acceleration);
    //! Check for move destination command
    bool get_destination_command(void);
    //! Issue move destination direct command
    void set_destination_direct(std::shared_ptr<Destination> destination, REAL velocity, REAL acceleration);
    //! Check for move destination direct command
    bool get_destination_direct_command(void);
    //! Get the destination commanded
    std::shared_ptr<Destination> get_destination(void);
    //! Get the waypoint commanded
    std::weak_ptr<Waypoint> get_waypoint(void);
    //! Set aborted status
    void set_aborted(void);
    //! Get aborted status
    bool get_aborted(void);
    //! Set error
    void set_error(DINT error);
    //! Get error status
    bool get_error(void);
    //! Get error id
    DINT get_error_id(void);
    //! Set move complete
    void set_move_done(void);
    //! Get move complete
    bool get_move_done(void);
    //! Set move active
    void set_move_active(void);
    //! Reset move active
    void reset_move_active(void);
    //! Get move active
    bool get_move_active(void);
    //! Set delete
    void set_delete(void);
    //! Get delete
    bool get_delete(void);
    //! Get velocity
    REAL get_velocity(void);
    //! Get acceleration
    REAL get_acceleration(void);
    //! Get existing shared pointer
    std::shared_ptr<ShuttleIf> get_shared_ptr(void);

    private:

    //! type identifier to ensure that pointer is valid
    UDINT _type_id = rl6dSHUTTLE_IF_TYPE_ID;
    //! Command Aborted
    bool _aborted = 0;
    //! Error
    bool _error = 0;
    //! Error ID
    DINT _error_id = 0;
    //! Move Destination
    bool _move_destination = 0;
    //! Move Destination Direct
    bool _move_destination_direct = 0;
    //! Destination
    std::shared_ptr<Destination> _destination;
    //! Route Waypoint
    std::weak_ptr<Waypoint> _waypoint;
    //! Velocity
    REAL _velocity;
    //! Acceleration
    REAL _acceleration;
    //! Move Done
    bool _move_done = 0;
    //! Move active
    bool _move_active = 0;
    //! Delete interface
    bool _delete = 0;

};

#endif
```

#### CheckRef.cpp - Check Reference Implementation
```cpp
#include "CheckRef.hpp"

DINT check_null_reference(UDINT reference){
    if(reference == 0){
        return rl6dERR_NULL_POINTER;
    }
    else{
        return ERR_OK;
    }
}

DINT check_router_reference(rl6dRouterType* reference){
    if(reference == nullptr){
        return rl6dERR_NULL_POINTER;
    }
    if(check_null_reference(reference->Ident) == ERR_OK){
        Router* router = reinterpret_cast<Router*>(reference->Ident);
        if(router->get_type_id() == rl6dROUTER_TYPE_ID){
            return ERR_OK;
        }
        else{
            return rl6dERR_ROUTER_INVALID;
        }
    }
    else{
        return rl6dERR_ROUTER_INVALID;
    }
}

DINT check_sem_man_reference(UDINT reference){
    DINT error;
    SemMan* sem_man;
    error = check_null_reference(reference);
    if(error == ERR_OK){
        sem_man = reinterpret_cast<SemMan*>(reference);
        if(sem_man->get_type_id() != rl6dSEM_MAN_TYPE_ID){
            error = rl6dERR_SEM_MAN_INVALID;
        }
    }
    return error;
}

DINT check_router_sem_reference(UDINT reference){
    DINT error;
    RouterSem* router_sem;
    error = check_null_reference(reference);
    if(error == ERR_OK){
        router_sem = reinterpret_cast<RouterSem*>(reference);
        if(router_sem->get_type_id() != rl6dROUTER_SEM_TYPE_ID){
            error = rl6dERR_ROUTER_SEM_INVALID;
        }
    }
    return error;
}

DINT check_destination_reference(rl6dDestinationType* reference){
    if(reference == nullptr){
        return rl6dERR_NULL_POINTER;
    }
    if(check_null_reference(reference->Ident) == ERR_OK){
        Destination* destination = reinterpret_cast<Destination*>(reference->Ident);
        if(destination->get_type_id() == rl6dDESTINATION_TYPE_ID){
            return ERR_OK;
        }
        else{
            return rl6dERR_DESTINATION_INVALID;
        }
    }
    else{
        return rl6dERR_DESTINATION_INVALID;
    }
}

DINT check_destination_if_reference(UDINT reference){
    DINT error;
    DestinationIf* destination_if;
    error = check_null_reference(reference);
    if(error == ERR_OK){
        destination_if = reinterpret_cast<DestinationIf*>(reference);
        if(destination_if->get_type_id() != rl6dDESTINATION_IF_TYPE_ID){
            error = rl6dERR_DESTINATION_IF_INVALID;
        }
    }
    return error;
}

DINT check_path_reference(rl6dPathType* reference){
    if(reference == nullptr){
        return rl6dERR_NULL_POINTER;
    }
    if(check_null_reference(reference->Ident) == ERR_OK){
        Path* path = reinterpret_cast<Path*>(reference->Ident);
        if(path->get_type_id() == rl6dPATH_TYPE_ID){
            return ERR_OK;
        }
        else{
            return rl6dERR_PATH_INVALID;
        }
    }
    else{
        return rl6dERR_PATH_INVALID;
    }
}

DINT check_waypoint_reference(rl6dWaypointType* reference){
    if(reference == nullptr){
        return rl6dERR_NULL_POINTER;
    }
    if(check_null_reference(reference->Ident) == ERR_OK){
        Waypoint* waypoint = reinterpret_cast<Waypoint*>(reference->Ident);
        if(waypoint->get_type_id() == rl6dWAYPOINT_TYPE_ID){
            return ERR_OK;
        }
        else{
            return rl6dERR_WAYPOINT_INVALID;
        }
    }
    else{
        return rl6dERR_WAYPOINT_INVALID;
    }
}

DINT check_shuttle_reference(rl6dShuttleType* reference){
    if(reference == nullptr){
        return rl6dERR_NULL_POINTER;
    }
    if(check_null_reference(reference->Ident) == ERR_OK){
        Shuttle* shuttle = reinterpret_cast<Shuttle*>(reference->Ident);
        if(shuttle->get_type_id() == rl6dSHUTTLE_TYPE_ID){
            return ERR_OK;
        }
        else{
            return rl6dERR_SHUTTLE_INVALID;
        }
    }
    else{
        return rl6dERR_SHUTTLE_INVALID;
    }
}

DINT check_shuttle_if_reference(UDINT reference){
    DINT error;
    ShuttleIf* shuttle_if;
    error = check_null_reference(reference);
    if(error == ERR_OK){
        shuttle_if = reinterpret_cast<ShuttleIf*>(reference);
        if(shuttle_if->get_type_id() != rl6dSHUTTLE_IF_TYPE_ID){
            error = rl6dERR_SHUTTLE_IF_INVALID;
        }
    }
    return error;
}
```

#### Logging.cpp - Logging Implementation
```cpp
#include "logging.hpp"

plcstring router_6d_log_name [] = "rl6dLog";

UDINT rl6d_log_buffer_min_size = 40;
UDINT rl6d_log_buffer_size_udint = 5;

bool log_routed_move_start(UINT shuttle, std::string destination){

    struct ArEventLogGetIdent get_ident;
    struct ArEventLogWrite write;

    bool status;
    UDINT buffer_size = destination.length() + 1;
    buffer_size += rl6d_log_buffer_min_size + rl6d_log_buffer_size_udint;
    char buffer [buffer_size];
    status = ArEventLogAddDataInit(reinterpret_cast<UDINT>(buffer), buffer_size, arEVENTLOG_ADDFORMAT_CODED);
    if(status){
        status = ArEventLogAddDataUdint(reinterpret_cast<UDINT>(buffer), buffer_size, shuttle);
    }
    if(status){
        status = ArEventLogAddDataString(reinterpret_cast<UDINT>(buffer), buffer_size, reinterpret_cast<UDINT>(destination.c_str()));
    }

    std::memset(&get_ident, 0, sizeof(get_ident));

    std::strcpy(get_ident.Name, router_6d_log_name);
    get_ident.Execute = 0;

    if(status){
        ArEventLogGetIdent(&get_ident);
        get_ident.Execute = 1;
        ArEventLogGetIdent(&get_ident);
        status = get_ident.Done;
        if(!status){
            get_ident.Execute = 0;
            ArEventLogGetIdent(&get_ident);
        }
    }

    std::memset(&write, 0, sizeof(write));

    std::string object = "RouterShuttle";
    object.append(std::to_string(shuttle));

    write.Ident = get_ident.Ident;
    std::strcpy(reinterpret_cast<char*>(&write.ObjectID), object.c_str());
    write.EventID = rl6dINFO_ROUTED_MOVE_START;
    write.AddData = reinterpret_cast<UDINT>(buffer);
    write.AddDataFormat = arEVENTLOG_ADDFORMAT_CODED;
    write.Execute = 0;

    if(status){
        ArEventLogWrite(&write);
        write.Execute = 1;
        ArEventLogWrite(&write);
        status = write.Done;
        write.Execute = 0;
        ArEventLogWrite(&write);
        get_ident.Execute = 0;
        ArEventLogGetIdent(&get_ident);
    }

    return status;

}

bool log_direct_move_start(UINT shuttle, std::string destination){

    struct ArEventLogGetIdent get_ident;
    struct ArEventLogWrite write;

    bool status;
    UDINT buffer_size = destination.length() + 1;
    buffer_size += rl6d_log_buffer_min_size + rl6d_log_buffer_size_udint;
    char buffer [buffer_size];
    status = ArEventLogAddDataInit(reinterpret_cast<UDINT>(buffer), buffer_size, arEVENTLOG_ADDFORMAT_CODED);
    if(status){
        status = ArEventLogAddDataUdint(reinterpret_cast<UDINT>(buffer), buffer_size, shuttle);
    }
    if(status){
        status = ArEventLogAddDataString(reinterpret_cast<UDINT>(buffer), buffer_size, reinterpret_cast<UDINT>(destination.c_str()));
    }

    std::memset(&get_ident, 0, sizeof(get_ident));

    std::strcpy(get_ident.Name, router_6d_log_name);
    get_ident.Execute = 0;

    if(status){
        ArEventLogGetIdent(&get_ident);
        get_ident.Execute = 1;
        ArEventLogGetIdent(&get_ident);
        status = get_ident.Done;
        if(!status){
            get_ident.Execute = 0;
            ArEventLogGetIdent(&get_ident);
        }
    }

    std::memset(&write, 0, sizeof(write));

    std::string object = "RouterShuttle";
    object.append(std::to_string(shuttle));

    write.Ident = get_ident.Ident;
    std::strcpy(reinterpret_cast<char*>(&write.ObjectID), object.c_str());
    write.EventID = rl6dINFO_DIRECT_MOVE_START;
    write.AddData = reinterpret_cast<UDINT>(buffer);
    write.AddDataFormat = arEVENTLOG_ADDFORMAT_CODED;
    write.Execute = 0;

    if(status){
        ArEventLogWrite(&write);
        write.Execute = 1;
        ArEventLogWrite(&write);
        status = write.Done;
        write.Execute = 0;
        ArEventLogWrite(&write);
        get_ident.Execute = 0;
        ArEventLogGetIdent(&get_ident);
    }

    return status;

}

bool log_destination_arrival(UINT shuttle, std::string destination){

    struct ArEventLogGetIdent get_ident;
    struct ArEventLogWrite write;

    bool status;
    UDINT buffer_size = destination.length() + 1;
    buffer_size += rl6d_log_buffer_min_size + rl6d_log_buffer_size_udint;
    char buffer [buffer_size];
    status = ArEventLogAddDataInit(reinterpret_cast<UDINT>(buffer), buffer_size, arEVENTLOG_ADDFORMAT_CODED);
    if(status){
        status = ArEventLogAddDataUdint(reinterpret_cast<UDINT>(buffer), buffer_size, shuttle);
    }
    if(status){
        status = ArEventLogAddDataString(reinterpret_cast<UDINT>(buffer), buffer_size, reinterpret_cast<UDINT>(destination.c_str()));
    }

    std::memset(&get_ident, 0, sizeof(get_ident));

    std::strcpy(get_ident.Name, router_6d_log_name);
    get_ident.Execute = 0;

    if(status){
        ArEventLogGetIdent(&get_ident);
        get_ident.Execute = 1;
        ArEventLogGetIdent(&get_ident);
        status = get_ident.Done;
        if(!status){
            get_ident.Execute = 0;
            ArEventLogGetIdent(&get_ident);
        }
    }

    std::memset(&write, 0, sizeof(write));

    std::string object = "RouterShuttle";
    object.append(std::to_string(shuttle));

    write.Ident = get_ident.Ident;
    std::strcpy(reinterpret_cast<char*>(&write.ObjectID), object.c_str());
    write.EventID = rl6dINFO_DESTINATION_ARRIVE;
    write.AddData = reinterpret_cast<UDINT>(buffer);
    write.AddDataFormat = arEVENTLOG_ADDFORMAT_CODED;
    write.Execute = 0;

    if(status){
        ArEventLogWrite(&write);
        write.Execute = 1;
        ArEventLogWrite(&write);
        status = write.Done;
        write.Execute = 0;
        ArEventLogWrite(&write);
        get_ident.Execute = 0;
        ArEventLogGetIdent(&get_ident);
    }

    return status;

}

bool log_destination_update(UINT shuttle, std::string destination){

    struct ArEventLogGetIdent get_ident;
    struct ArEventLogWrite write;

    bool status;
    UDINT buffer_size = destination.length() + 1;
    buffer_size += rl6d_log_buffer_min_size + rl6d_log_buffer_size_udint;
    char buffer [buffer_size];
    status = ArEventLogAddDataInit(reinterpret_cast<UDINT>(buffer), buffer_size, arEVENTLOG_ADDFORMAT_CODED);
    if(status){
        status = ArEventLogAddDataUdint(reinterpret_cast<UDINT>(buffer), buffer_size, shuttle);
    }
    if(status){
        status = ArEventLogAddDataString(reinterpret_cast<UDINT>(buffer), buffer_size, reinterpret_cast<UDINT>(destination.c_str()));
    }

    std::memset(&get_ident, 0, sizeof(get_ident));

    std::strcpy(get_ident.Name, router_6d_log_name);
    get_ident.Execute = 0;

    if(status){
        ArEventLogGetIdent(&get_ident);
        get_ident.Execute = 1;
        ArEventLogGetIdent(&get_ident);
        status = get_ident.Done;
        if(!status){
            get_ident.Execute = 0;
            ArEventLogGetIdent(&get_ident);
        }
    }

    std::memset(&write, 0, sizeof(write));

    std::string object = "RouterShuttle";
    object.append(std::to_string(shuttle));

    write.Ident = get_ident.Ident;
    std::strcpy(reinterpret_cast<char*>(&write.ObjectID), object.c_str());
    write.EventID = rl6dINFO_DESTINATION_UPDATE;
    write.AddData = reinterpret_cast<UDINT>(buffer);
    write.AddDataFormat = arEVENTLOG_ADDFORMAT_CODED;
    write.Execute = 0;

    if(status){
        ArEventLogWrite(&write);
        write.Execute = 1;
        ArEventLogWrite(&write);
        status = write.Done;
        write.Execute = 0;
        ArEventLogWrite(&write);
        get_ident.Execute = 0;
        ArEventLogGetIdent(&get_ident);
    }

    return status;

}

bool log_path_start(UINT shuttle, std::string path){

    struct ArEventLogGetIdent get_ident;
    struct ArEventLogWrite write;

    bool status;
    UDINT buffer_size = path.length() + 1;
    buffer_size += rl6d_log_buffer_min_size + rl6d_log_buffer_size_udint;
    char buffer [buffer_size];
    status = ArEventLogAddDataInit(reinterpret_cast<UDINT>(buffer), buffer_size, arEVENTLOG_ADDFORMAT_CODED);
    if(status){
        status = ArEventLogAddDataUdint(reinterpret_cast<UDINT>(buffer), buffer_size, shuttle);
    }
    if(status){
        status = ArEventLogAddDataString(reinterpret_cast<UDINT>(buffer), buffer_size, reinterpret_cast<UDINT>(path.c_str()));
    }

    std::memset(&get_ident, 0, sizeof(get_ident));

    std::strcpy(get_ident.Name, router_6d_log_name);
    get_ident.Execute = 0;

    if(status){
        ArEventLogGetIdent(&get_ident);
        get_ident.Execute = 1;
        ArEventLogGetIdent(&get_ident);
        status = get_ident.Done;
        if(!status){
            get_ident.Execute = 0;
            ArEventLogGetIdent(&get_ident);
        }
    }

    std::memset(&write, 0, sizeof(write));

    std::string object = "RouterShuttle";
    object.append(std::to_string(shuttle));

    write.Ident = get_ident.Ident;
    std::strcpy(reinterpret_cast<char*>(&write.ObjectID), object.c_str());
    write.EventID = rl6dINFO_MOVE_PATH_START;
    write.AddData = reinterpret_cast<UDINT>(buffer);
    write.AddDataFormat = arEVENTLOG_ADDFORMAT_CODED;
    write.Execute = 0;

    if(status){
        ArEventLogWrite(&write);
        write.Execute = 1;
        ArEventLogWrite(&write);
        status = write.Done;
        write.Execute = 0;
        ArEventLogWrite(&write);
        get_ident.Execute = 0;
        ArEventLogGetIdent(&get_ident);
    }

    return status;

}

bool log_waypoint_move(UINT shuttle, std::string waypoint){

    struct ArEventLogGetIdent get_ident;
    struct ArEventLogWrite write;

    bool status;
    UDINT buffer_size = waypoint.length() + 1;
    buffer_size += rl6d_log_buffer_min_size + rl6d_log_buffer_size_udint;
    char buffer [buffer_size];
    status = ArEventLogAddDataInit(reinterpret_cast<UDINT>(buffer), buffer_size, arEVENTLOG_ADDFORMAT_CODED);
    if(status){
        status = ArEventLogAddDataUdint(reinterpret_cast<UDINT>(buffer), buffer_size, shuttle);
    }
    if(status){
        status = ArEventLogAddDataString(reinterpret_cast<UDINT>(buffer), buffer_size, reinterpret_cast<UDINT>(waypoint.c_str()));
    }

    std::memset(&get_ident, 0, sizeof(get_ident));

    std::strcpy(get_ident.Name, router_6d_log_name);
    get_ident.Execute = 0;

    if(status){
        ArEventLogGetIdent(&get_ident);
        get_ident.Execute = 1;
        ArEventLogGetIdent(&get_ident);
        status = get_ident.Done;
        if(!status){
            get_ident.Execute = 0;
            ArEventLogGetIdent(&get_ident);
        }
    }

    std::memset(&write, 0, sizeof(write));

    std::string object = "RouterShuttle";
    object.append(std::to_string(shuttle));

    write.Ident = get_ident.Ident;
    std::strcpy(reinterpret_cast<char*>(&write.ObjectID), object.c_str());
    write.EventID = rl6dINFO_MOVE_WAYPOINT;
    write.AddData = reinterpret_cast<UDINT>(buffer);
    write.AddDataFormat = arEVENTLOG_ADDFORMAT_CODED;
    write.Execute = 0;

    if(status){
        ArEventLogWrite(&write);
        write.Execute = 1;
        ArEventLogWrite(&write);
        status = write.Done;
        write.Execute = 0;
        ArEventLogWrite(&write);
        get_ident.Execute = 0;
        ArEventLogGetIdent(&get_ident);
    }

    return status;

}

bool log_asm_get_sh_start(){

    struct ArEventLogGetIdent get_ident;
    struct ArEventLogWrite write;

    bool status;

    std::memset(&get_ident, 0, sizeof(get_ident));

    std::strcpy(get_ident.Name, router_6d_log_name);
    get_ident.Execute = 0;

    ArEventLogGetIdent(&get_ident);
    get_ident.Execute = 1;
    ArEventLogGetIdent(&get_ident);
    status = get_ident.Done;
    if(!status){
        get_ident.Execute = 0;
        ArEventLogGetIdent(&get_ident);
    }

    std::memset(&write, 0, sizeof(write));

    write.Ident = get_ident.Ident;
    std::strcpy(reinterpret_cast<char*>(&write.ObjectID), "Router");
    write.EventID = rl6dINFO_GET_SHUTTLES_START;
    write.Execute = 0;

    if(status){
        ArEventLogWrite(&write);
        write.Execute = 1;
        ArEventLogWrite(&write);
        status = write.Done;
        write.Execute = 0;
        ArEventLogWrite(&write);
        get_ident.Execute = 0;
        ArEventLogGetIdent(&get_ident);
    }

    return status;

}
bool log_asm_get_sh_done(UINT shuttles){

    struct ArEventLogGetIdent get_ident;
    struct ArEventLogWrite write;

    bool status;
    UDINT buffer_size = rl6d_log_buffer_min_size + rl6d_log_buffer_size_udint;
    char buffer [buffer_size];
    status = ArEventLogAddDataInit(reinterpret_cast<UDINT>(buffer), buffer_size, arEVENTLOG_ADDFORMAT_CODED);
    if(status){
        status = ArEventLogAddDataUdint(reinterpret_cast<UDINT>(buffer), buffer_size, shuttles);
    }

    std::memset(&get_ident, 0, sizeof(get_ident));

    std::strcpy(get_ident.Name, router_6d_log_name);
    get_ident.Execute = 0;

    if(status){
        ArEventLogGetIdent(&get_ident);
        get_ident.Execute = 1;
        ArEventLogGetIdent(&get_ident);
        status = get_ident.Done;
        if(!status){
            get_ident.Execute = 0;
            ArEventLogGetIdent(&get_ident);
        }
    }

    std::memset(&write, 0, sizeof(write));

    write.Ident = get_ident.Ident;
    std::strcpy(reinterpret_cast<char*>(&write.ObjectID), "Router");
    write.EventID = rl6dINFO_GET_SHUTTLES_DONE;
    write.AddData = reinterpret_cast<UDINT>(buffer);
    write.AddDataFormat = arEVENTLOG_ADDFORMAT_CODED;
    write.Execute = 0;

    if(status){
        ArEventLogWrite(&write);
        write.Execute = 1;
        ArEventLogWrite(&write);
        status = write.Done;
        write.Execute = 0;
        ArEventLogWrite(&write);
        get_ident.Execute = 0;
        ArEventLogGetIdent(&get_ident);
    }

    return status;

}

bool log_asm_recovery_start(rl6dRecoverModeEnum mode){

    struct ArEventLogGetIdent get_ident;
    struct ArEventLogWrite write;

    bool status;
    UDINT buffer_size = rl6d_log_buffer_min_size + rl6d_log_buffer_size_udint;
    char buffer [buffer_size];
    status = ArEventLogAddDataInit(reinterpret_cast<UDINT>(buffer), buffer_size, arEVENTLOG_ADDFORMAT_CODED);
    if(status){
        status = ArEventLogAddDataDint(reinterpret_cast<UDINT>(buffer), buffer_size, mode);
    }

    std::memset(&get_ident, 0, sizeof(get_ident));

    std::strcpy(get_ident.Name, router_6d_log_name);
    get_ident.Execute = 0;

    if(status){
        ArEventLogGetIdent(&get_ident);
        get_ident.Execute = 1;
        ArEventLogGetIdent(&get_ident);
        status = get_ident.Done;
        if(!status){
            get_ident.Execute = 0;
            ArEventLogGetIdent(&get_ident);
        }
    }

    std::memset(&write, 0, sizeof(write));

    write.Ident = get_ident.Ident;
    std::strcpy(reinterpret_cast<char*>(&write.ObjectID), "Router");
    write.EventID = rl6dINFO_RECOVERY_START;
    write.AddData = reinterpret_cast<UDINT>(buffer);
    write.AddDataFormat = arEVENTLOG_ADDFORMAT_CODED;
    write.Execute = 0;

    if(status){
        ArEventLogWrite(&write);
        write.Execute = 1;
        ArEventLogWrite(&write);
        status = write.Done;
        write.Execute = 0;
        ArEventLogWrite(&write);
        get_ident.Execute = 0;
        ArEventLogGetIdent(&get_ident);
    }

    return status;

}
bool log_asm_recovery_done(void){

    struct ArEventLogGetIdent get_ident;
    struct ArEventLogWrite write;

    bool status;

    std::memset(&get_ident, 0, sizeof(get_ident));

    std::strcpy(get_ident.Name, router_6d_log_name);
    get_ident.Execute = 0;

    ArEventLogGetIdent(&get_ident);
    get_ident.Execute = 1;
    ArEventLogGetIdent(&get_ident);
    status = get_ident.Done;
    if(!status){
        get_ident.Execute = 0;
        ArEventLogGetIdent(&get_ident);
    }

    std::memset(&write, 0, sizeof(write));

    write.Ident = get_ident.Ident;
    std::strcpy(reinterpret_cast<char*>(&write.ObjectID), "Router");
    write.EventID = rl6dINFO_RECOVERY_DONE;
    write.Execute = 0;

    if(status){
        ArEventLogWrite(&write);
        write.Execute = 1;
        ArEventLogWrite(&write);
        status = write.Done;
        write.Execute = 0;
        ArEventLogWrite(&write);
        get_ident.Execute = 0;
        ArEventLogGetIdent(&get_ident);
    }

    return status;
}
bool log_asm_sh_assignment(UINT shuttle, std::string destination){

    struct ArEventLogGetIdent get_ident;
    struct ArEventLogWrite write;

    bool status;
    UDINT buffer_size = destination.length() + 1;
    buffer_size += rl6d_log_buffer_min_size + rl6d_log_buffer_size_udint;
    char buffer [buffer_size];
    status = ArEventLogAddDataInit(reinterpret_cast<UDINT>(buffer), buffer_size, arEVENTLOG_ADDFORMAT_CODED);
    if(status){
        status = ArEventLogAddDataUdint(reinterpret_cast<UDINT>(buffer), buffer_size, shuttle);
    }
    if(status){
        status = ArEventLogAddDataString(reinterpret_cast<UDINT>(buffer), buffer_size, reinterpret_cast<UDINT>(destination.c_str()));
    }

    std::memset(&get_ident, 0, sizeof(get_ident));

    std::strcpy(get_ident.Name, router_6d_log_name);
    get_ident.Execute = 0;

    if(status){
        ArEventLogGetIdent(&get_ident);
        get_ident.Execute = 1;
        ArEventLogGetIdent(&get_ident);
        status = get_ident.Done;
        if(!status){
            get_ident.Execute = 0;
            ArEventLogGetIdent(&get_ident);
        }
    }

    std::memset(&write, 0, sizeof(write));

    write.Ident = get_ident.Ident;
    std::strcpy(reinterpret_cast<char*>(&write.ObjectID), "Router");
    write.EventID = rl6dINFO_RECOVERY_ASSIGNMENT;
    write.AddData = reinterpret_cast<UDINT>(buffer);
    write.AddDataFormat = arEVENTLOG_ADDFORMAT_CODED;
    write.Execute = 0;

    if(status){
        ArEventLogWrite(&write);
        write.Execute = 1;
        ArEventLogWrite(&write);
        status = write.Done;
        write.Execute = 0;
        ArEventLogWrite(&write);
        get_ident.Execute = 0;
        ArEventLogGetIdent(&get_ident);
    }

    return status;

}
bool log_sh_error(UINT shuttle, DINT error){

    struct ArEventLogGetIdent get_ident;
    struct ArEventLogWrite write;

    bool status;
    UDINT buffer_size = rl6d_log_buffer_min_size + (rl6d_log_buffer_size_udint * 2);
    char buffer [buffer_size];
    status = ArEventLogAddDataInit(reinterpret_cast<UDINT>(buffer), buffer_size, arEVENTLOG_ADDFORMAT_CODED);
    if(status){
        status = ArEventLogAddDataUdint(reinterpret_cast<UDINT>(buffer), buffer_size, shuttle);
    }
    if(status){
        status = ArEventLogAddDataDint(reinterpret_cast<UDINT>(buffer), buffer_size, error);
    }

    std::memset(&get_ident, 0, sizeof(get_ident));

    std::strcpy(get_ident.Name, router_6d_log_name);
    get_ident.Execute = 0;

    if(status){
        ArEventLogGetIdent(&get_ident);
        get_ident.Execute = 1;
        ArEventLogGetIdent(&get_ident);
        status = get_ident.Done;
        if(!status){
            get_ident.Execute = 0;
            ArEventLogGetIdent(&get_ident);
        }
    }

    std::memset(&write, 0, sizeof(write));

    std::string object = "RouterShuttle";
    object.append(std::to_string(shuttle));

    write.Ident = get_ident.Ident;
    std::strcpy(reinterpret_cast<char*>(&write.ObjectID), object.c_str());
    write.EventID = rl6dERR_SHUTTLE;
    write.AddData = reinterpret_cast<UDINT>(buffer);
    write.AddDataFormat = arEVENTLOG_ADDFORMAT_CODED;
    write.Execute = 0;

    if(status){
        ArEventLogWrite(&write);
        write.Execute = 1;
        ArEventLogWrite(&write);
        status = write.Done;
        write.Execute = 0;
        ArEventLogWrite(&write);
        get_ident.Execute = 0;
        ArEventLogGetIdent(&get_ident);
    }

    return status;

}
bool log_asm_get_sh_error(DINT error){

    struct ArEventLogGetIdent get_ident;
    struct ArEventLogWrite write;

    bool status;
    UDINT buffer_size = rl6d_log_buffer_min_size + rl6d_log_buffer_size_udint;
    char buffer [buffer_size];
    status = ArEventLogAddDataInit(reinterpret_cast<UDINT>(buffer), buffer_size, arEVENTLOG_ADDFORMAT_CODED);
    if(status){
        status = ArEventLogAddDataDint(reinterpret_cast<UDINT>(buffer), buffer_size, error);
    }

    std::memset(&get_ident, 0, sizeof(get_ident));

    std::strcpy(get_ident.Name, router_6d_log_name);
    get_ident.Execute = 0;

    if(status){
        ArEventLogGetIdent(&get_ident);
        get_ident.Execute = 1;
        ArEventLogGetIdent(&get_ident);
        status = get_ident.Done;
        if(!status){
            get_ident.Execute = 0;
            ArEventLogGetIdent(&get_ident);
        }
    }

    std::memset(&write, 0, sizeof(write));

    write.Ident = get_ident.Ident;
    std::strcpy(reinterpret_cast<char*>(&write.ObjectID), "Router");
    write.EventID = rl6dERR_SHUTTLE;
    write.AddData = reinterpret_cast<UDINT>(buffer);
    write.AddDataFormat = arEVENTLOG_ADDFORMAT_CODED;
    write.Execute = 0;

    if(status){
        ArEventLogWrite(&write);
        write.Execute = 1;
        ArEventLogWrite(&write);
        status = write.Done;
        write.Execute = 0;
        ArEventLogWrite(&write);
        get_ident.Execute = 0;
        ArEventLogGetIdent(&get_ident);
    }

    return status;

}
bool log_move_in_plane_error(DINT error){

    struct ArEventLogGetIdent get_ident;
    struct ArEventLogWrite write;

    bool status;
    UDINT buffer_size = rl6d_log_buffer_min_size + rl6d_log_buffer_size_udint;
    char buffer [buffer_size];
    status = ArEventLogAddDataInit(reinterpret_cast<UDINT>(buffer), buffer_size, arEVENTLOG_ADDFORMAT_CODED);
    if(status){
        status = ArEventLogAddDataDint(reinterpret_cast<UDINT>(buffer), buffer_size, error);
    }

    std::memset(&get_ident, 0, sizeof(get_ident));

    std::strcpy(get_ident.Name, router_6d_log_name);
    get_ident.Execute = 0;

    if(status){
        ArEventLogGetIdent(&get_ident);
        get_ident.Execute = 1;
        ArEventLogGetIdent(&get_ident);
        status = get_ident.Done;
        if(!status){
            get_ident.Execute = 0;
            ArEventLogGetIdent(&get_ident);
        }
    }

    std::memset(&write, 0, sizeof(write));

    write.Ident = get_ident.Ident;
    std::strcpy(reinterpret_cast<char*>(&write.ObjectID), "Router");
    write.EventID = rl6dERR_SHUTTLE;
    write.AddData = reinterpret_cast<UDINT>(buffer);
    write.AddDataFormat = arEVENTLOG_ADDFORMAT_CODED;
    write.Execute = 0;

    if(status){
        ArEventLogWrite(&write);
        write.Execute = 1;
        ArEventLogWrite(&write);
        status = write.Done;
        write.Execute = 0;
        ArEventLogWrite(&write);
        get_ident.Execute = 0;
        ArEventLogGetIdent(&get_ident);
    }

    return status;

}
```

#### Router.cpp - Router Implementation
```cpp
#include "Router.hpp"

Router::Router(Mc6DAssemblyType* assembly, UDINT user_data_size){
    std::memset(&this->_asm_get_shuttle, 0, sizeof(this->_asm_get_shuttle));
    std::memset(&this->_move_in_plane_async, 0, sizeof(this->_move_in_plane_async));
    std::memset(&this->_ar_event_log_create, 0, sizeof(this->_ar_event_log_create));
    this->_asm_get_shuttle.Assembly = assembly;
    this->_move_in_plane_async.Assembly = assembly;
    this->_user_data_size = user_data_size;
}

//destructor
Router::~Router(){
    this->_type_id = rl6dNO_TYPE_ID;
}

// methods
UDINT Router::get_type_id(){
    return this->_type_id;
}
void Router::set_add_sh_from_asm(){
    this->_cmd.add_sh_from_asm = 1;
}
void Router::reset_add_sh_from_asm(){
    this->_cmd.add_sh_from_asm = 0;
}
void Router::set_error_reset(){
    this->_cmd.error_reset = 1;
}
UINT Router::get_num_asm_sh(){
    return this->_asm_shuttles;
}
void Router::set_recover_shuttles(rl6dRecoverModeEnum mode, REAL velocity, REAL acceleration){
    this->_move_in_plane_async.Parameters.Velocity = velocity;
    this->_move_in_plane_async.Parameters.Acceleration = acceleration;
    this->_cmd.recover_shuttles_mode = mode;
    this->_cmd.recover_shuttles = 1;
}
void Router::reset_recover_shuttles(){
    this->_cmd.recover_shuttles = 0;
    this->_cmd.recover_shuttles_mode = rl6dRECOVER_MODE_BASIC;
}
bool Router::get_cmd_ready(){
    return this->_status.cmd_ready;
}
bool Router::get_done(){
    return this->_status.done;
}
std::shared_ptr<Path> Router::create_path(std::string name, std::shared_ptr<RouterSem> router_sem){
    auto it = std::find_if(this->_paths.begin(), this->_paths.end(), [name](std::shared_ptr<Path> i){return i->get_name() == name;});
    if(it == this->_paths.end()){
        std::shared_ptr<Path> path (new Path(name, router_sem));
        this->_paths.push_back(path);
        return path;
    }
    else{
        throw std::invalid_argument("Path with given name already exists.");
    }
}
std::shared_ptr<Destination> Router::create_destination(std::string name, std::shared_ptr<RouterSem> router_sem, rl6dPositionType position, std::shared_ptr<Path> path_in, std::shared_ptr<Path> path_out){
    auto it = std::find_if(this->_destinations.begin(), this->_destinations.end(), [name](std::shared_ptr<Destination> i){return i->get_name() == name;});
        if(it == this->_destinations.end()){
        std::shared_ptr<Destination> destination (new Destination(name, router_sem, position, path_in, path_out));
        this->_destinations.push_back(destination);
        return destination;
    }
    else{
        throw std::invalid_argument("Destination with given name already exists.");
    }
}
std::shared_ptr<Waypoint> Router::create_waypoint(std::string name, std::shared_ptr<RouterSem> router_sem, rl6dPositionType position){
    auto it = std::find_if(this->_waypoints.begin(), this->_waypoints.end(), [name](std::shared_ptr<Waypoint> i){return i->get_name() == name;});
        if(it == this->_waypoints.end()){
        std::shared_ptr<Waypoint> waypoint (new Waypoint(name, router_sem, position));
        this->_waypoints.push_back(waypoint);
        return waypoint;
    }
    else{
        throw std::invalid_argument("Waypoint with given name already exists.");
    }
}
void Router::delete_path(std::shared_ptr<Path> path){
    auto it = std::find_if(this->_paths.begin(), this->_paths.end(), [path](std::shared_ptr<Path> i){return i == path;});
    if(it == this->_paths.end()){
        throw std::invalid_argument("Path not defined in Router.");
    }
    else{
        this->_paths.erase(it);
    }
}
std::shared_ptr<Path> Router::get_path_by_name(std::string name){

    auto it = std::find_if(this->_paths.begin(), this->_paths.end(), [name](std::shared_ptr<Path> i){return i->get_name() == name;});
    if(it == this->_paths.end()){
        throw std::invalid_argument("Path with given name does not exist.");
    }
    else{
        return *it;
    }
}
std::shared_ptr<Shuttle> Router::add_shuttle(Mc6DShuttleType shuttle, std::shared_ptr<RouterSem> router_semaphore, UINT shuttle_id){
    for (auto & existing_shuttle : this->_shuttles){
        if (existing_shuttle->get_shuttle_reference()->controlif == shuttle.controlif){
            throw std::invalid_argument("Shuttle already in router.");
        }
    }
    std::shared_ptr<Shuttle> routed_shuttle (new Shuttle(shuttle, router_semaphore, this->_user_data_size, shuttle_id));
    this->_shuttles.push_back(routed_shuttle);
    return routed_shuttle;
}
bool Router::acquire_path_semaphore(){
    return this->_path_semaphore->sem_acquire();
}
void Router::release_path_semaphore(){
    this->_path_semaphore->sem_release();
}
bool Router::acquire_waypoint_semaphore(){
    return this->_waypoint_semaphore->sem_acquire();
}
void Router::release_waypoint_semaphore(){
    this->_waypoint_semaphore->sem_release();
}
bool Router::acquire_shuttle_semaphore(){
    return this->_shuttle_semaphore->sem_acquire();
}
void Router::release_shuttle_semaphore(){
    this->_shuttle_semaphore->sem_release();
}
bool Router::acquire_destination_semaphore(){
    return this->_destination_semaphore->sem_acquire();
}
void Router::release_destination_semaphore(){
    this->_destination_semaphore->sem_release();
}
bool Router::acquire_cmd_semaphore(){
    return this->_command_semaphore->sem_acquire();
}
void Router::release_cmd_semaphore(){
    this->_command_semaphore->sem_release();
}
bool Router::get_initialized(){
    return this->_init_done;
}
bool Router::get_error(){
    return this->_error;
}
DINT Router::get_error_id(){
    return this->_error_id;
}
void Router::cyclic(){

    bool done;

    switch(this->_state){

        case STATE_INIT:

            std::strcpy(this->_ar_event_log_create.Name, router_6d_log_name);
            this->_ar_event_log_create.Size = 10000; //TODO
            this->_ar_event_log_create.Persistence = arEVENTLOG_PERSISTEN CE_PERSIST; //TODO
            this->_ar_event_log_create.Execute = 1;
            this->_state = STATE_EVENT_LOG_CREATE;

            break;

        case STATE_EVENT_LOG_CREATE:

            if(this->_ar_event_log_create.Done || this->_ar_event_log_create.Error){
                this->_ar_event_log_create.Execute = 0;
                this->_state = STATE_WAIT_SEM;
            }

            break;

        case STATE_WAIT_SEM:

            if(this->_semaphore_manager.get_initialized()){
                if(this->sem_acquire()){
                    if(this->get_sem_cmd_ready()){
                        this->set_create_sem();
                        this->_state = STATE_CREATE_PATH_SEM;
                    }
                    else{
                        this->sem_release();
                    }
                }
            }

            break;

        case STATE_CREATE_PATH_SEM:

            if(this->get_sem_done()){
                this->_path_semaphore = this->get_created_sem();
                this->reset_create_sem();
                this->_state = STATE_CREATE_WAYPOINT_SEM_READY;
            }

            break;

        case STATE_CREATE_WAYPOINT_SEM_READY:

            if(this->get_sem_cmd_ready()){
                this->set_create_sem();
                this->_state = STATE_CREATE_WAYPOINT_SEM;
            }

            break;

        case STATE_CREATE_WAYPOINT_SEM:

            if(this->get_sem_done()){
                this->_waypoint_semaphore = this->get_created_sem();
                this->reset_create_sem();
                this->_state = STATE_CREATE_SHUTTLE_SEM_READY;
            }

            break;

        case STATE_CREATE_SHUTTLE_SEM_READY:

            if(this->get_sem_cmd_ready()){
                this->set_create_sem();
                this->_state = STATE_CREATE_SHUTTLE_SEM;
            }

            break;

        case STATE_CREATE_SHUTTLE_SEM:

            if(this->get_sem_done()){
                this->_shuttle_semaphore = this->get_created_sem();
                this->reset_create_sem();
                this->_state = STATE_CREATE_DESTINATION_SEM_READY;
            }

            break;

        case STATE_CREATE_DESTINATION_SEM_READY:

            if(this->get_sem_cmd_ready()){
                this->set_create_sem();
                this->_state = STATE_CREATE_DESTINATION_SEM;
            }

            break;

        case STATE_CREATE_DESTINATION_SEM:

            if(this->get_sem_done()){
                this->_destination_semaphore = this->get_created_sem();
                this->reset_create_sem();
                this->_state = STATE_CREATE_CMD_SEM_READY;
            }

            break;

        case STATE_CREATE_CMD_SEM_READY:

            if(this->get_sem_cmd_ready()){
                this->set_create_sem();
                this->_state = STATE_CREATE_CMD_SEM;
            }

        break;

        case STATE_CREATE_CMD_SEM:

            if(this->get_sem_done()){
                this->_command_semaphore = this->get_created_sem();
                this->reset_create_sem();
                this->sem_release();
                this->_init_done = 1;
                this->_status.cmd_ready = 1;
                this->_state = STATE_ACTIVE;
            }

        break;

        case STATE_ACTIVE:

            this->_router_sem_complete = 1;
            if(this->_cmd.add_sh_from_asm){
                log_asm_get_sh_start();
                this->_status.cmd_ready = 0;
                this->_old_remaining_count = 0;
                this->_asm_get_shuttle.Enable = 1;
                this->_state = STATE_ADD_SH_ASM;
            }
            else if(this->_cmd.recover_shuttles){
                if(this->acquire_shuttle_semaphore()){
                    log_asm_recovery_start(this->_cmd.recover_shuttles_mode);
                    this->_recovery_shuttles = this->_shuttles;
                    this->release_shuttle_semaphore();
                    this->_status.cmd_ready = 0;
                    this->_state = STATE_RECOVER_SHUTTLES_GET_DEST;
                }
            }

            break;

        case STATE_ADD_SH_ASM:

            if(this->_asm_get_shuttle.Error){
                log_asm_get_sh_error(this->_asm_get_shuttle.ErrorID);
                this->_asm_get_shuttle.Next = 0;
                this->_asm_get_shuttle.Enable = 0;
                this->_error_id = this->_asm_get_shuttle.ErrorID;
                this->_shuttles.clear();
                this->_state = STATE_ERROR;
            }
            else if(this->_asm_get_shuttle.Valid){
                if(this->_asm_get_shuttle.TotalCount == 0){
                    this->_status.done = 1;
                    log_asm_get_sh_done(this->_asm_get_shuttle.TotalCount);
                    this->_asm_shuttles = 0;
                    this->_state = STATE_ADD_SH_ASM_DONE;
                }
                else if((this->_asm_get_shuttle.RemainingCount != this->_old_remaining_count) || (this->_asm_get_shuttle.TotalCount == 1)){
                    this->_asm_get_shuttle.Next = 0;
                        if(this->sem_acquire()){
                        if(this->get_sem_cmd_ready()){
                            this->set_create_sem();
                            this->_state = STATE_ADD_SH_ASM_SEM;
                        }
                        else{
                            this->sem_release();
                        }
                    }
                }
            }

            break;

        case STATE_ADD_SH_ASM_SEM:

            if(this->get_sem_done()){
                this->_created_semaphore = this->get_created_sem();
                this->reset_create_sem();
                this->sem_release();
                this->_state = STATE_ADD_SH_ASM_NEXT;
            }

            break;

        case STATE_ADD_SH_ASM_NEXT:

            if(this->acquire_shuttle_semaphore()){
                this->add_shuttle(this->_asm_get_shuttle.Shuttle, this->_created_semaphore, this->_asm_get_shuttle.AdditionalInfo.ShuttleID);
                this->release_shuttle_semaphore();
                this->_created_semaphore.reset();
                if(this->_asm_get_shuttle.RemainingCount == 0){
                    log_asm_get_sh_done(this->_asm_get_shuttle.TotalCount);
                    this->_asm_get_shuttle.Enable = 0;
                    this->_asm_shuttles = this->_asm_get_shuttle.TotalCount;
                    this->_status.done = 1;
                    this->_state = STATE_ADD_SH_ASM_DONE;
                }
                else{
                    this->_old_remaining_count = this->_asm_get_shuttle.RemainingCount;
                    this->_asm_get_shuttle.Next = 1;
                    this->_state = STATE_ADD_SH_ASM;
                }
            }

            break;

        case STATE_ADD_SH_ASM_DONE:

            if(!this->_cmd.add_sh_from_asm){
                this->_asm_shuttles = 0;
                this->_status.done = 0;
                this->_status.cmd_ready = 1;
                this->_state = STATE_ACTIVE;
            }

            break;

        case STATE_RECOVER_SHUTTLES_GET_DEST:

            if(this->acquire_destination_semaphore()){
                this->_recovery_destinations = this->_destinations;
                this->release_destination_semaphore();
                if(this->_recovery_destinations.empty()){
                    this->_status.done = 1;
                    log_asm_recovery_done();
                    this->_state = STATE_RECOVER_SHUTTLES_DONE;
                }
                else{
                    this->_current_recovery_destination = this->_recovery_destinations.back();
                    this->_recovery_destinations.pop_back();
                    this->_current_recovery_index = 0;
                    this->_state = STATE_RECOVER_SHUTTLES_GET_POS;
                }
            }

            break;

        case STATE_RECOVER_SHUTTLES_GET_POS:

            if(this->_current_recovery_destination->sem_acquire()){
                this->_current_recovery_positions = this->_current_recovery_destination->get_recovery_positions();
                this->_current_recovery_destination->sem_release();
                this->_state = STATE_RECOVER_SHUTTLES_ASSIGN;
            }

            break;

        case STATE_RECOVER_SHUTTLES_ASSIGN:

            while(this->_current_recovery_index < rl6dMAX_RECOVER_SHUTTLES){
                if(this->_recovery_shuttles.empty()){
                    break;
                }
                if(this->_current_recovery_positions.empty()){
                    break;
                }
                this->_current_recovery_shuttle = this->_recovery_shuttles.back();
                log_asm_sh_assignment(this->_current_recovery_shuttle->get_shuttle_id(), this->_current_recovery_destination->get_name());
                this->_shuttle_destination_assignment.push_back(ShDestAssignment{this->_current_recovery_shuttle, this->_current_recovery_destination});
                this->_recovery_shuttles.pop_back();
                this->_current_recovery_position = this->_current_recovery_positions.back();
                this->_current_recovery_positions.pop_back();
                this->_move_in_plane_async.Parameters.AsyncPar[this->_current_recovery_index].Shuttle = this->_current_recovery_shuttle->get_shuttle_reference();
                this->_move_in_plane_async.Parameters.AsyncPar[this->_current_recovery_index].X = this->_current_recovery_position.X;
                this->_move_in_plane_async.Parameters.AsyncPar[this->_current_recovery_index].Y = this->_current_recovery_position.Y;
                this->_current_recovery_index++;
            }
            if(this->_recovery_shuttles.empty()){
                //All shuttles have been assigned
                if(this->_current_recovery_index > 0){
                    //There is at least one shuttle to recover
                    this->_move_in_plane_async.Execute = 1;
                    this->_state = STATE_RECOVER_SHUTTLES;
                }
                else{
                    //There are no shuttles to recover
                    this->_recovery_destinations.clear();
                    this->_current_recovery_positions.clear();
                    this->_current_recovery_shuttle.reset();
                    this->_current_recovery_destination.reset();
                    this->_state = STATE_RECOVER_DESTINATION;
                }
            }
            else if(this->_current_recovery_index >= (rl6dMAX_RECOVER_SHUTTLES - 1)){
                //The Async function block has all indices assigned
                this->_move_in_plane_async.Execute = 1;
                this->_state = STATE_RECOVER_SHUTTLES;
            }
            else{
                //We are out of recovery positions on this destination
                if(this->_recovery_destinations.empty()){
                    if(this->_current_recovery_index > 0){
                        //There is at least one position we can recover to
                        this->_move_in_plane_async.Execute = 1;
                        this->_state = STATE_RECOVER_SHUTTLES;
                    }
                    else{
                        //There are no positions we can recover to
                        this->_recovery_shuttles.clear();
                        this->_current_recovery_positions.clear();
                        this->_current_recovery_shuttle.reset();
                        this->_current_recovery_destination.reset();
                        this->_state = STATE_RECOVER_DESTINATION;
                    }
                }
                else{
                    this->_current_recovery_destination = this->_recovery_destinations.back();
                    this->_recovery_destinations.pop_back();
                    this->_state = STATE_RECOVER_SHUTTLES_GET_POS;
                }
            }

            break;

        case STATE_RECOVER_SHUTTLES:

            if(this->_move_in_plane_async.Done){
                this->_move_in_plane_async.Execute = 0;
                this->_current_recovery_index = 0;
                this->_state = STATE_RECOVER_SHUTTLES_ASSIGN;
            }
            else if(this->_move_in_plane_async.Error){
                log_move_in_plane_error(this->_move_in_plane_async.ErrorID);
                this->_move_in_plane_async.Execute = 0;
                this->_status.error_id = this->_move_in_plane_async.ErrorID;
                this->_status.error = 1;
                this->_state = STATE_ERROR;
            }

            break;

        case STATE_RECOVER_DESTINATION:

            while(!this->_shuttle_destination_assignment.empty()){
                this->_current_recovery_shuttle = this->_shuttle_destination_assignment.back().shuttle;
                this->_current_recovery_destination = this->_shuttle_destination_assignment.back().destination;
                if(this->_current_recovery_shuttle->sem_acquire()){
                    this->_current_recovery_shuttle_interface = this->_current_recovery_shuttle->create_interface();

                    this->_current_recovery_shuttle_interface->set_destination_direct(this->_current_recovery_destination,
                                                                                      this->_move_in_plane_async.Parameters.Velocity,
                                                                                      this->_move_in_plane_async.Parameters.Acceleration);

                this->_shuttle_recovery_interfaces.push_back(this->_current_recovery_shuttle_interface);
                    this->_shuttle_destination_assignment.pop_back();
                    this->_current_recovery_shuttle->sem_release();
                }
                else{
                    break;
                }
            }
            if(this->_shuttle_destination_assignment.empty()){
                this->_current_recovery_shuttle.reset();
                this->_current_recovery_destination.reset();
                this->_current_recovery_shuttle_interface.reset();
                this->_state = STATE_RECOVER_DESTINATION_WAIT;
            }

            break;

        case STATE_RECOVER_DESTINATION_WAIT:

            done = 1;
            for(auto & interface : this->_shuttle_recovery_interfaces){
                if(interface->get_type_id() == rl6dSHUTTLE_IF_TYPE_ID){
                    if(interface->get_error()){
                        this->_status.error_id = interface->get_error_id();
                        this->_status.error = 1;
                        for(auto & interface : this->_shuttle_recovery_interfaces){
                            if(interface->get_type_id() == rl6dSHUTTLE_IF_TYPE_ID){
                                interface->set_delete();
                            }
                        }
                        this->_shuttle_recovery_interfaces.clear();
                        this->_state = STATE_ERROR;
                        break;
                    }
                    else if(!(interface->get_move_active() || interface->get_move_done() || interface->get_aborted())){
                        done = 0;
                    }
                }
                //TODO: Add handling for if the list of interfaces contains an invalid interface
            }
            if(done){
                for(auto & interface : this->_shuttle_recovery_interfaces){
                    if(interface->get_type_id() == rl6dSHUTTLE_IF_TYPE_ID){
                        interface->set_delete();
                    }
                }
                this->_shuttle_recovery_interfaces.clear();
                this->_status.done = 1;
                log_asm_recovery_done();
                this->_state = STATE_RECOVER_SHUTTLES_DONE;
            }

            break;

        case STATE_RECOVER_SHUTTLES_DONE:

            if(!this->_cmd.recover_shuttles){
                this->_status.done = 0;
                this->_status.cmd_ready = 1;
                this->_state = STATE_ACTIVE;
            }

            break;

        case STATE_ERROR:

            this->_error = 1;
            if(this->_cmd.error_reset){
                this->_error_id = ERR_OK;
                this->_error = 0;
            }

            break;

    }

    this->_semaphore_manager.cyclic();
    if(this->_router_sem_complete){
        if(this->acquire_shuttle_semaphore()){
            for(auto & shuttle : this->_shuttles){
                shuttle->cyclic();
            }
            this->release_shuttle_semaphore();
        }
        if(this->acquire_destination_semaphore()){
            for(auto & destination : this->_destinations){
                destination->cyclic();
            }
            this->release_destination_semaphore();
        }
    }
    MC_BR_AsmGetShuttle_Acp6D(&this->_asm_get_shuttle);
    MC_BR_MoveInPlaneAsync_Acp6D(&this->_move_in_plane_async);
    ArEventLogCreate(&this->_ar_event_log_create);

    this->_cmd.error_reset = 0;

}
```
